(* IEC 61131-3 sources: OpenPLC_v3/webserver/st_files, 2 files *)

(* ---- 331092.st ---- *)
PROGRAM NoOperation
  VAR
    unused_var: BOOL;
  END_VAR
  unused_var:=FALSE;
END_PROGRAM
CONFIGURATION Config0
  RESOURCE Res0 ON PLC
    TASK IdleTask(INTERVAL := T#100ms, PRIORITY := 1);
    PROGRAM IdleInstance WITH IdleTask : NoOperation;
  END_RESOURCE
END_CONFIGURATION

(* ---- blank_program.st ---- *)
PROGRAM prog0
  VAR
    var_in : BOOL;
    var_out : BOOL;
  END_VAR

  var_out := var_in;
END_PROGRAM

CONFIGURATION Config0

  RESOURCE Res0 ON PLC
    TASK Main(INTERVAL := T#50ms,PRIORITY := 0);
    PROGRAM Inst0 WITH Main : prog0;
  END_RESOURCE
END_CONFIGURATION
